// TIA Portal V18 export
VAR_GLOBAL   // PLC tag table "Cabinet_11"
   Sz11_ST13_SenA AT %I2100.0 : Bool;
   Sz11_ST13_SenB AT %I2100.1 : Bool;
   Sz11_ST13_SenC AT %I2100.2 : Bool;
   Sz11_ST13_SenD AT %I2100.3 : Bool;
   Sz11_ST14_SenA AT %I2100.4 : Bool;
   Sz11_ST14_SenB AT %I2100.5 : Bool;
   Sz11_ST14_SenC AT %I2100.6 : Bool;
   Sz11_ST14_SenD AT %I2100.7 : Bool;
   Sz11_ST17_SenA AT %I2101.0 : Bool;
   Sz11_ST17_SenB AT %I2101.1 : Bool;
   Sz11_ST17_SenC AT %I2101.2 : Bool;
   Sz11_ST17_SenD AT %I2101.3 : Bool;
   "Reserved(188)" AT %I2101.4 : Bool;
   "Reserved(189)" AT %I2101.5 : Bool;
   "Reserved(190)" AT %I2101.6 : Bool;
   Sz11_Safety1_1 AT %I2150.0 : Bool;
   "Reserved(173)" AT %I2150.1 : Bool;
   "Reserved(174)" AT %I2150.2 : Bool;
   "Reserved(175)" AT %I2150.3 : Bool;
   Sz11_Safety1_2 AT %I2150.4 : Bool;
   "Reserved(176)" AT %I2150.5 : Bool;
   "Reserved(177)" AT %I2150.6 : Bool;
   "Reserved(178)" AT %I2150.7 : Bool;
   "Reserved(179)" AT %I2151.0 : Bool;
   "Reserved(180)" AT %I2151.1 : Bool;
   "Reserved(181)" AT %I2151.2 : Bool;
   "Reserved(182)" AT %I2151.3 : Bool;
   "Reserved(183)" AT %I2151.4 : Bool;
   "Reserved(184)" AT %I2151.5 : Bool;
   "Reserved(185)" AT %I2151.6 : Bool;
   "Reserved(186)" AT %I2151.7 : Bool;
   Sz11_Button_LED_ST13_ST14 AT %Q2100.0 : Bool;
   "Reserved(187)" AT %I2101.7 : Bool;
   Sz11_Button_LED_SS_Down AT %Q2100.1 : Bool;
   Sz11_Button_LED_SS_Up AT %Q2100.2 : Bool;
   Sz11_Button_LED_SS_Drive_ST14 AT %Q2100.3 : Bool;
   Sz11_Button_LED_SS_Drive_ST17 AT %Q2100.4 : Bool;
   Sz11_Button_LED_SS_Drive_ST24 AT %Q2100.5 : Bool;
   Sz11_Button_LED_SS_Drive_ST25 AT %Q2100.6 : Bool;
   "Reserved(172)" AT %Q2100.7 : Bool;
   Sz11_Button_ST13_ST14 AT %I2102.0 : Bool;
   Sz11_Button_SS_Down AT %I2102.1 : Bool;
   Sz11_Button_SS_Up AT %I2102.2 : Bool;
   Sz11_Button_SS_Drive_ST14 AT %I2102.3 : Bool;
   Sz11_Button_SS_Drive_ST17 AT %I2102.4 : Bool;
   Sz11_Button_SS_Drive_ST24 AT %I2102.5 : Bool;
   Sz11_Button_SS_Drive_ST25 AT %I2102.6 : Bool;
END_VAR
